FUNCTION Get_Vel_RPM : DINT
VAR_INPUT
	Increment_Per_Sec : DINT := 0;
END_VAR

Get_Vel_RPM := (Increment_Per_Sec/4096) * 60;

END_FUNCTION

(* stored: Version 1.1.0.1, ProductVersion 3.1.4024.12
   POU Get_Vel_RPM: Id {23e05a45-c99c-453e-bf0b-883758330c29}, SpecialFunc None *)
